{attribute addProperty BoxType "EK1960-0000-0019"}
{attribute addProperty Id "FSOEAT %I*FSOE_F3ED5C6B12015"}
{attribute addProperty CRC "4275424613"}
{attribute addProperty SizeInBites "120"}
{attribute addProperty SizeInBytes "15"}
TYPE FSoE_Inputs_FED5CD65 :
STRUCT
	{attribute addProperty Name "FSOE"}
	FSOE AT %I* : FSOE_F3ED5C6B;
END_STRUCT
END_TYPE

(* stored: Version 1.2.0.0, ProductVersion 3.1.4024.9
   DUT FSoE_Inputs_FED5CD65: Id {45113c80-fe69-4174-bba5-7543e66f9a3a} *)
